FUNCTION EngUnits_to_MeasureUnit : REAL
VAR_INPUT
	rValue		: REAL;
	rSlope 		: REAL;
	rOffset 	: REAL;
END_VAR
VAR
END_VAR

MeasureUnit_to_EngUnits := (rValue*rSlope)+rOffset;

END_FUNCTION

(* stored: Version 1.1.0.1, ProductVersion 3.1.4024.12
   POU EngUnits_to_MeasureUnit: Id {1bc54788-5d73-4be0-b261-d23d606f36ae}, SpecialFunc None *)
